{attribute 'qualified_only'}
VAR_GLOBAL
	//ADD COVER SERVO AND STEPPER MOTOR TO SOLUTION
	servoBackward AT %Q*: BOOL := FALSE;
	servoForward AT %Q*: BOOL := false;
END_VAR

(* stored: Version 1.1.0.1, ProductVersion 3.1.4024.5
   GVL DSout: Id {7006bbd0-77a0-4d8c-b300-1141a8c09454} *)
